Fanuc KAREL source: ka00143.KL

PROGRAM KA00143
%NOLOCKGROUP
VAR
SRC : ARRAY[2] OF SHORT
DST : ARRAY[2] OF BYTE
BEGIN
SRC[1]=2
DST[1]=SRC[1]
END KA00143
